{attribute 'qualified_only'}
{attribute 'strict'}
{attribute 'to_string'}
TYPE TYPE_CATEGORY :
(
    VALUE_TYPE := 0,
	REFERENCE_TYPE := 1
) BYTE;
END_TYPE

(* stored: Version 1.1.0.1
   DUT TYPE_CATEGORY: Id {38457657-3233-48a9-8ff1-e662e036e2ba} *)
